PROGRAM MAIN
VAR
	State 			: INT	:=0  ;

	ToTimeoutbool 	: TON ;
	T1Timer 		: BOOL ;
	enable 			: BOOL;
	rTrigenable 	: R_TRIG;
END_VAR

rTrigenable(CLk := enable);
ToTimeoutbool(IN := T1Timer,PT := T#2S);
IF gvl.Morning THEN
	state := 0;
END_IF
	CASE state OF
	0:
		GVL.WakeUp 					:= TRUE;
		T1Timer 					:= TRUE;
		IF ToTimeoutbool.Q THEN
			T1Timer 				:= FALSE;
			GVL.WakeUp 				:= FALSE ;
			state := 1; 
		END_IF
		
	1:
		GVL.MakeTheBed 				:= TRUE;
			T1Timer 				:= TRUE;
		IF ToTimeoutbool.Q THEN
			T1Timer 				:= FALSE;
			GVL.MakeTheBed 			:= FALSE ;
			state := 2;
		END_IF
		
	2:
		GVL.TakeShower 				:= TRUE;
		T1Timer 					:= TRUE;
		IF ToTimeoutbool.Q THEN
			T1Timer := FALSE;
			GVL.TakeShower 			:= FALSE ;
			state := 3;
		END_IF
		
	3:
		GVL.DateCheck				:= TRUE;
		State := 4; 

	4: 
		IF gvl.Day = 'Sat' OR gvl.Day = 'Sun' THEN
			routine2();
			gvl.SRoutine2 			:= TRUE;
			State					:= 5;
		ELSIF gvl.Day = 'Weekdays' THEN
		 	routine1();		
			GVl.SRoutine1 			:= TRUE ;
			State					:= 5;
		END_IF
	5:
		gvl.Morning 				:= FALSE;
	
		
	END_CASE

END_PROGRAM

(* stored: Version 1.1.0.1, ProductVersion 3.1.4024.12
   POU MAIN: Id {5eeb6e1b-3578-49b3-8f85-ec5f5e749d55}, SpecialFunc None *)
